{region '#Template'}
	{attribute 'Version' := '5.3.0.0'}
	{attribute 'Tags' := '"LCID": "1031", "Text": "Fassade, Sonnenschutz"'}
	{attribute 'Tags' := '"LCID": "1033", "Text": "Facade, Sunprotection"'}
	{attribute 'Using' := '"Type": "Template", "URI": "Site"'}
	{attribute 'Using' := '"Type": "Template", "URI": "ST_BA_Facade"'}
	{attribute 'Description' := '"LCID": "1031", "Text": "Sonnenschutz Fassadendaten"'}
	{attribute 'Description' := '"LCID": "1033", "Text": "Sunprotection facade data"'}
{endregion}
// General fascade template:
// - Calculation and distribution of fascade information
FUNCTION_BLOCK FB_BA_Facade EXTENDS FB_BA_View
VAR_INPUT
	fRefRmT			: REAL;
	fRefRmTCol		: REAL;
	fRefRmTHtg		: REAL;
END_VAR
VAR_OUTPUT
	stFacade		: ST_BA_Facade;
END_VAR

VAR_INPUT CONSTANT PERSISTENT
	{attribute 'parameterUnit':= 'deg'}
	fFcdOrtn					: REAL;		// orientation [deg] of the facade
	{attribute 'parameterUnit':= 'deg'}
	fFcdAngl					: REAL;		// declination [deg] of the facade
	{attribute 'parameterUnit':= 'mm'}
	fLamWdth					: REAL;		// lamella width [mm]
	{attribute 'parameterUnit':= 'mm'}
	fLamDstc					: REAL;		// space between two lamellas [mm]
                                      
	{attribute 'parameterUnit':= 'deg'}
	fAzmSttRng					: REAL;		// azimuth start-range [deg] when facade is in sun
	{attribute 'parameterUnit':= 'deg'}
	fAzmEndRng					: REAL;		// azimuth end-range [deg] when facade is in sun
	{attribute 'parameterUnit':= 'deg'}
	fElvLoLmt					: REAL;		// elevation start-range [deg] when facade is in sun
	{attribute 'parameterUnit':= 'deg'}
	fElvHiLmt					: REAL;		// elevation end-range [deg] when facade is in sun
END_VAR

VAR_INPUT CONSTANT
	CommError					: FB_BA_SunBldEvt			:=(ePrio:=E_BA_SunBldPrio.eCommError);	
	WindProtection				: FB_BA_Facade_WindProtection;
	Maintenance					: FB_BA_Facade_Maintenance;
	ThermoAutomatic				: FB_BA_Facade_ThermoAutomatic;
	TwilightAutomatic			: FB_BA_Facade_TwilightAutomatic;
	ParkPosition				: FB_BA_Facade_ParkPosition;
	SunProtection				: FB_BA_Facade_SunProtection;
	FacadeInformation			: FB_BA_Facade_Information;
END_VAR	

VAR			
	InRngAzm					: FB_BA_InRngAzm;
	InRngElv					: FB_BA_InRngElv;
	bFcdInSun					: BOOL;	
	SunBldTgmResult				: FB_BA_SunBldTgmSel8;	
END_VAR
VAR // added by the converter: edge detectors and wires of the graphical bodies
    _s1 : ST_BA_Facade;
    _w1 : BOOL;
END_VAR

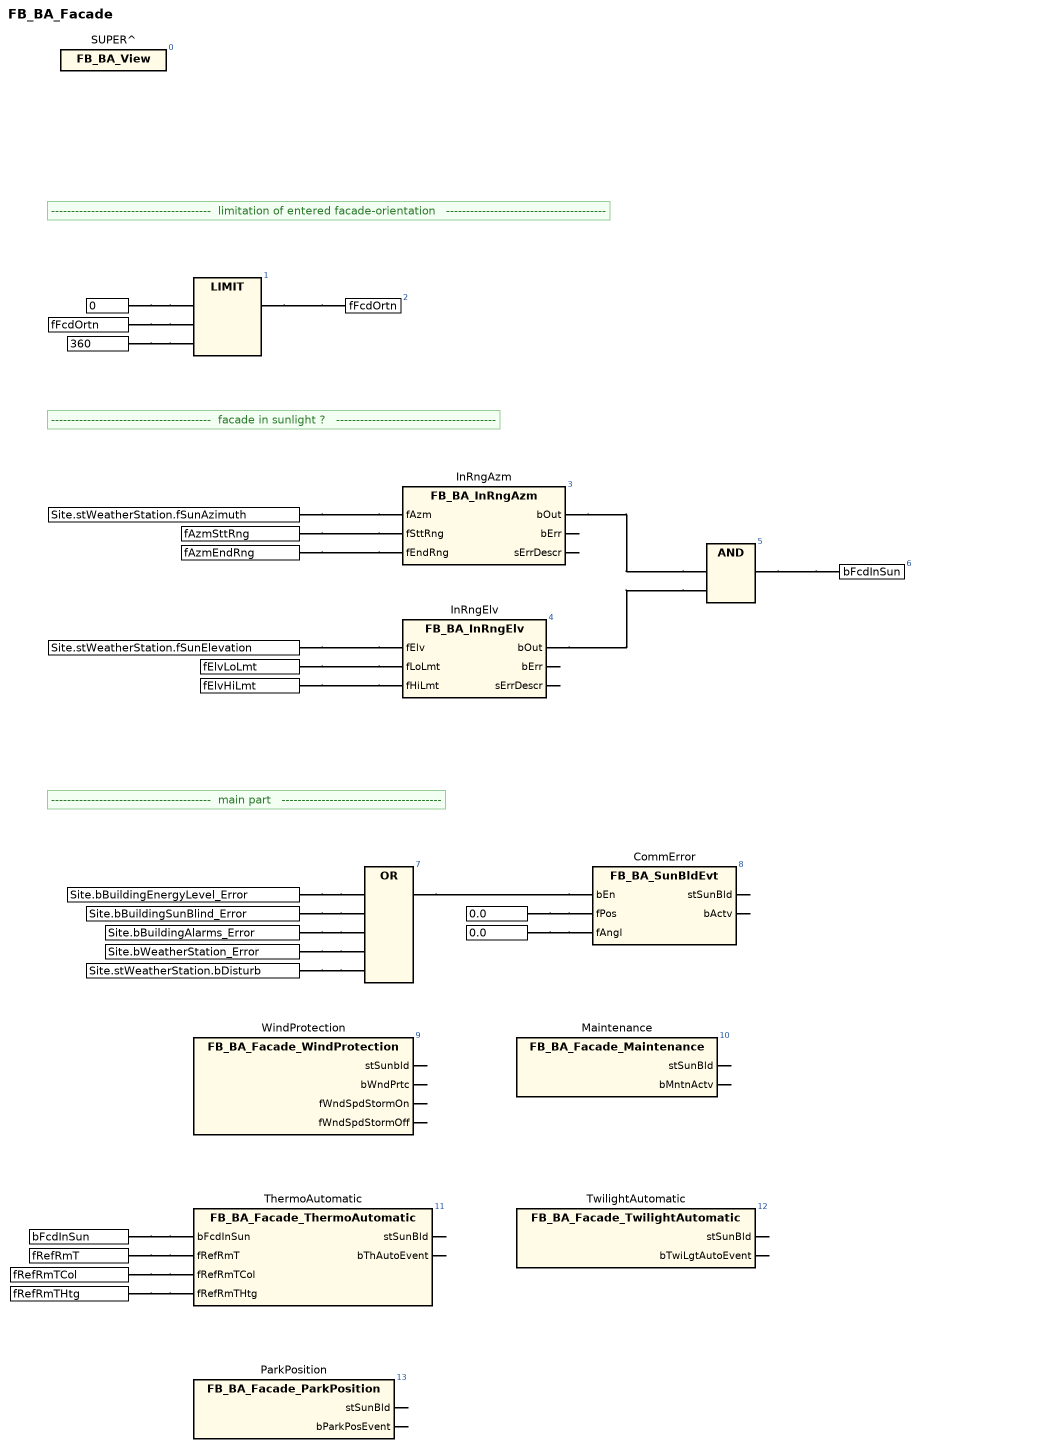
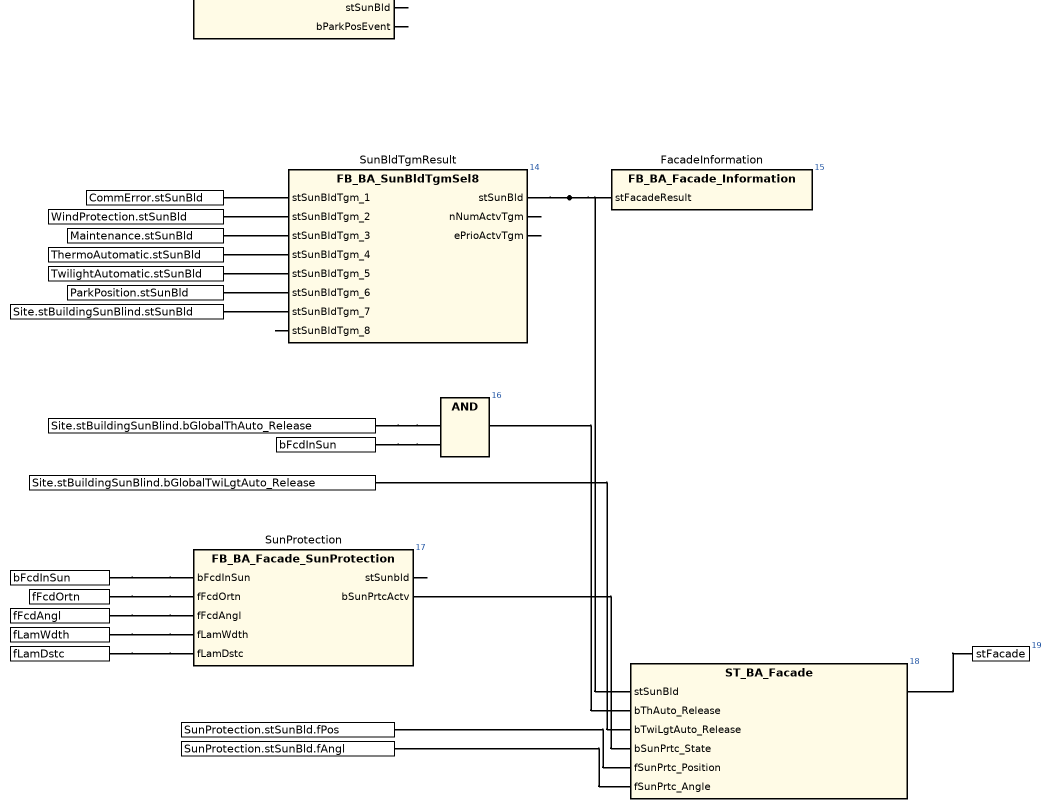
SUPER^(); // FB_BA_View
// ----------------------------------------  limitation of entered facade-orientation   ----------------------------------------
fFcdOrtn := LIMIT(0, fFcdOrtn, 360);
// ----------------------------------------  facade in sunlight ?   ----------------------------------------
InRngAzm(fAzm := Site.stWeatherStation.fSunAzimuth, fSttRng := fAzmSttRng, fEndRng := fAzmEndRng); // FB_BA_InRngAzm
InRngElv(fElv := Site.stWeatherStation.fSunElevation, fLoLmt := fElvLoLmt, fHiLmt := fElvHiLmt); // FB_BA_InRngElv
bFcdInSun := InRngAzm.bOut AND InRngElv.bOut;
// ----------------------------------------  main part   ----------------------------------------
CommError(
    bEn := Site.bBuildingEnergyLevel_Error OR Site.bBuildingSunBlind_Error OR Site.bBuildingAlarms_Error OR Site.bWeatherStation_Error OR Site.stWeatherStation.bDisturb,
    fPos := 0.0,
    fAngl := 0.0); // FB_BA_SunBldEvt
WindProtection(); // FB_BA_Facade_WindProtection
Maintenance(); // FB_BA_Facade_Maintenance
ThermoAutomatic(
    bFcdInSun := bFcdInSun,
    fRefRmT := fRefRmT,
    fRefRmTCol := fRefRmTCol,
    fRefRmTHtg := fRefRmTHtg); // FB_BA_Facade_ThermoAutomatic
TwilightAutomatic(); // FB_BA_Facade_TwilightAutomatic
ParkPosition(); // FB_BA_Facade_ParkPosition
SunBldTgmResult(
    stSunBldTgm_1 := CommError.stSunBld,
    stSunBldTgm_2 := WindProtection.stSunBld,
    stSunBldTgm_3 := Maintenance.stSunBld,
    stSunBldTgm_4 := ThermoAutomatic.stSunBld,
    stSunBldTgm_5 := TwilightAutomatic.stSunBld,
    stSunBldTgm_6 := ParkPosition.stSunBld,
    stSunBldTgm_7 := Site.stBuildingSunBlind.stSunBld); // FB_BA_SunBldTgmSel8
FacadeInformation(stFacadeResult := SunBldTgmResult.stSunBld); // FB_BA_Facade_Information
_w1 := Site.stBuildingSunBlind.bGlobalThAuto_Release AND bFcdInSun;
SunProtection(
    bFcdInSun := bFcdInSun,
    fFcdOrtn := fFcdOrtn,
    fFcdAngl := fFcdAngl,
    fLamWdth := fLamWdth,
    fLamDstc := fLamDstc); // FB_BA_Facade_SunProtection
// compose _s1 : ST_BA_Facade
_s1.stSunBld := SunBldTgmResult.stSunBld;
_s1.bThAuto_Release := _w1;
_s1.bTwiLgtAuto_Release := Site.stBuildingSunBlind.bGlobalTwiLgtAuto_Release;
_s1.bSunPrtc_State := SunProtection.bSunPrtcActv;
_s1.fSunPrtc_Position := SunProtection.stSunBld.fPos;
_s1.fSunPrtc_Angle := SunProtection.stSunBld.fAngl;
stFacade := _s1;

METHOD FB_init : BOOL
VAR_INPUT
	bInitRetains : BOOL; // if TRUE; the retain variables are initialized (warm start / cold start)
	bInCopyCode : BOOL;  // if TRUE; the instance afterwards gets moved into the copy code (online change)
END_VAR

VAR

END_VAR
WindProtection.iParent				:= THIS^;	
WindProtection.iLabel				:= LblCtl_WindProtection;
WindProtection.sObjectName		   	:= '{Idx=01}';
WindProtection.eDPADMode			:= E_BA_DPADMode.eInclude;
                                                           
Maintenance.iParent					:= THIS^;	
Maintenance.iLabel					:= LblCtl_Maintenance;
Maintenance.sObjectName		   		:= '{Idx=01}';
Maintenance.eDPADMode				:= E_BA_DPADMode.eInclude;
                            	                            	
ThermoAutomatic.iParent				:= THIS^;	
ThermoAutomatic.iLabel				:= LblCtl_ThermoAutomatic;
ThermoAutomatic.sObjectName		   	:= '{Idx=01}';
ThermoAutomatic.eDPADMode			:= E_BA_DPADMode.eInclude;                            	

TwilightAutomatic.iParent			:= THIS^;	
TwilightAutomatic.iLabel			:= LblCtl_TwilightAutomatic;
TwilightAutomatic.sObjectName		:= '{Idx=01}';
TwilightAutomatic.eDPADMode			:= E_BA_DPADMode.eInclude;     

ParkPosition.iParent				:= THIS^;	
ParkPosition.iLabel					:= LblCtl_Parking;
ParkPosition.sObjectName			:= '{Idx=01}';
ParkPosition.eDPADMode				:= E_BA_DPADMode.eInclude;     

SunProtection.iParent				:= THIS^;	
SunProtection.iLabel				:= LblCtl_SunProtection;
SunProtection.sObjectName			:= '{Idx=01}';
SunProtection.eDPADMode				:= E_BA_DPADMode.eInclude;     

FacadeInformation.iParent			:= THIS^;	
FacadeInformation.iLabel			:= LblCtl_FacadeInformation;
FacadeInformation.sObjectName		:= '{Idx=01}';
FacadeInformation.eDPADMode			:= E_BA_DPADMode.eInclude;
END_METHOD

END_FUNCTION_BLOCK

(* stored: Version 1.1.0.1, ProductVersion 3.1.4024.12
   POU FB_BA_Facade: Id {837c4797-0cfd-455c-b2c3-fb6cd568b568}, SpecialFunc None
   Method FB_init: Id {e3239c1a-b997-43f6-90c0-2e8755ef0a93} *)
